{attribute 'GeneratedUsingTerminal: EL2596-0000-0017'}
{attribute addProperty BoxType "EL2596-0000-0017"}
{attribute addProperty Id "EnableBOOL1OutputBOOL1Input_trigger_enableBOOL1Output_trigger_enableBOOL1ResetBOOL1"}
{attribute addProperty CRC "318348406"}
{attribute addProperty Size "5"}
TYPE Control_12F99C76 :
STRUCT
	{attribute addProperty Name "Enable"}
	Enable : BOOL;
	{attribute addProperty Name "Output"}
	Output : BOOL;
	{attribute addProperty Name "Input_trigger_enable"}
	Input_trigger_enable : BOOL;
	{attribute addProperty Name "Output_trigger_enable"}
	Output_trigger_enable : BOOL;
	{attribute addProperty Name "Reset"}
	Reset : BOOL;
END_STRUCT
END_TYPE

(* stored: Version 1.2.0.0, ProductVersion 3.1.4024.9
   DUT Control_12F99C76: Id {783a6a9f-d91a-46c1-b0fb-f8bd198f39e9} *)
